FUNCTION_BLOCK FB_IntensiveWash IMPLEMENTS I_WashStrategy
VAR
	stWashSettings : ST_WashSettings;
END_VAR

METHOD FB_init : BOOL
VAR_INPUT
	bInitRetains : BOOL; // if TRUE, the retain variables are initialized (warm start / cold start)
	bInCopyCode : BOOL;  // if TRUE, the instance afterwards gets moved into the copy code (online change)
END_VAR
IF stWashSettings.sDescription = '' THEN
	stWashSettings.rWashTemperature := GVL_WashConstants.INTENSIVE_TEMP;
	stWashSettings.nSpinSpeed:= GVL_WashConstants.INTENSIVE_SPIN;
	stWashSettings.tWashDuration := GVL_WashConstants.INTENSIVE_WASH_TIME;
	stWashSettings.sDescription := GVL_WashConstants.INTENSIVE_DESC;
	
END_IF
FB_init :=TRUE;
END_METHOD

{warning 'add method implementation '}
METHOD GetProgramName : STRING
GetProgramName := 'Intensive';
END_METHOD

METHOD GetRinseTime : TIME
VAR_INPUT
END_VAR
GetRinseTime := GVL_WashConstants.NORMAL_WASH_RINSE_TIME;
END_METHOD

METHOD GetSpinTime : TIME
VAR_INPUT
END_VAR
GetSpinTime := GVL_WashConstants.NORMAL_WASH_SPIN_TIME;
END_METHOD


METHOD GetWashSettings : ST_WashSettings
GetWashSettings := stWashSettings;
END_METHOD

END_FUNCTION_BLOCK

(* stored: Version 1.1.0.1, ProductVersion 3.1.4024.16
   POU FB_IntensiveWash: Id {1b624a9a-787a-46df-943d-ffbad20b2ca8}, SpecialFunc None
   Method FB_init: Id {65b911fa-e470-4825-9c70-7cbfa5837ab3}
   Method GetProgramName: Id {994d12cf-fbc6-45d2-883a-a099bfdf27c6}
   Method GetRinseTime: Id {15aa26cc-268e-4c0c-902b-1a09f828145a}
   Method GetSpinTime: Id {c61f6559-0b5f-4628-a4d5-ec64dceb2e68}
   Method GetWashSettings: Id {94ac178f-107e-4af5-9eb7-e84316509b2b} *)
